PROGRAM pouTestMessages
VAR
	i: INT;
	retvall: UDINT;
END_VAR
VAR // added by the converter: edge detectors and wires of the graphical bodies
    _rt1, _rt2 : R_TRIG;
END_VAR

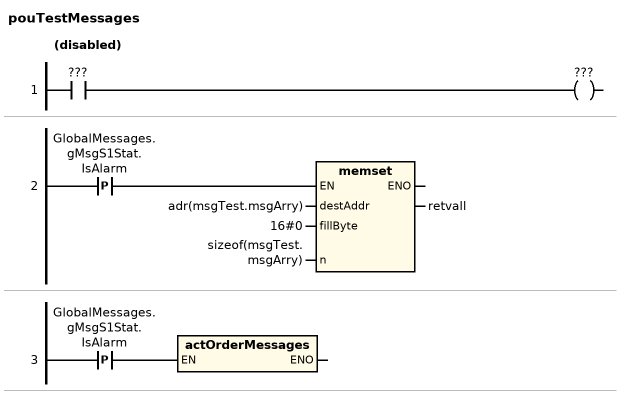
// NETWORK 1 (disabled)
// ??? := ???;

// NETWORK 2
_rt1(CLK := GlobalMessages.gMsgS1Stat.IsAlarm);
IF _rt1.Q THEN
    retvall := memset(destAddr := adr(msgTest.msgArry), fillByte := 16#0, n := sizeof(msgTest.msgArry));
END_IF

// NETWORK 3
_rt2(CLK := GlobalMessages.gMsgS1Stat.IsAlarm);
IF _rt2.Q THEN actOrderMessages(); END_IF

ACTION actOrderMessages:
FOR i:= 1 TO 100 DO

//GlobalMessages.gListMsgS1.AlarmViewMsg

//move message text
msgTest.msgArry[i].text := GlobalMessages.gListMsgS1.AlarmViewMsg[i].msgText;

//apply colour
msgTest.msgArryStyle[i].isColoured := GlobalMessages.gListMsgS1.AlarmViewMsg[i].isAlarm OR GlobalMessages.gListMsgS1.AlarmViewMsg[i].isWarning;

	//apply alarm colour
	IF  GlobalMessages.gListMsgS1.AlarmViewMsg[i].isAlarm  THEN
		msgTest.msgArryStyle[i].colourToApply := HMIColour.colourRed;
	END_IF

	IF  GlobalMessages.gListMsgS1.AlarmViewMsg[i].isWarning  THEN
		msgTest.msgArryStyle[i].colourToApply := HMIColour.colourYellow;
	END_IF
	
msgTest.msgArry[i].timeRaised := '12:30:32AM';
msgTest.msgArry[i].timeResolved := '13:30:32AM';

msgTest.msgArry[i].source := 'Station 1';



	
END_FOR
END_ACTION

END_PROGRAM

(* stored: Version 1.1.0.1, ProductVersion 3.1.4024.12
   POU pouTestMessages: Id {2f973ab8-75ab-4ca6-a5d1-6370fde62421}, SpecialFunc None
   Action actOrderMessages: Id {81b0e784-c3ff-42a5-87b7-d9bc89652420} *)
